{attribute 'qualified_only'}
{attribute 'strict'}
TYPE E_IOSensorType :
(
	NO 		:= 0,
	NC		:= 1,
	NOx2	:= 2
);
END_TYPE

(* stored: Version 1.1.0.1
   DUT E_IOSensorType: Id {7d151584-babf-4f04-a36d-c72d7215a9e8} *)
